% RSLogix 500 project PROC1_COUNTER_RESET_BAK001.RSS, saved by version 8.30.00.16 %
PROJECT "PROC1"    % processor: Bul.1763 MicroLogix 1100 Series B %

PROGRAM FILES
  LAD 2 "MAIN"  2 rungs
  LAD 3 "COUNTERS"  4 rungs

DATA FILES
  O0 OUTPUT  4 elements
  I1 INPUT  6 elements
  S2 STATUS  66 elements
  B3 BINARY  1 elements
  T4 TIMER  1 elements
  C5 COUNTER  1 elements
  R6 CONTROL  1 elements
  N7 INTEGER  1 elements
  F8 FLOAT  1 elements

LADDER 2 "MAIN"
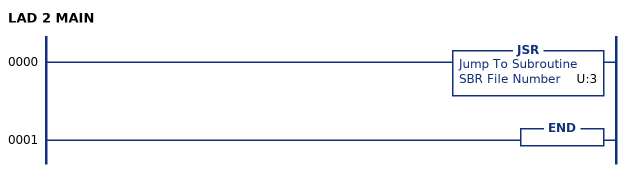
% Rung: 0 %
SOR JSR U:3 EOR
% Rung: 1 %
SOR END EOR

LADDER 3 "COUNTERS"
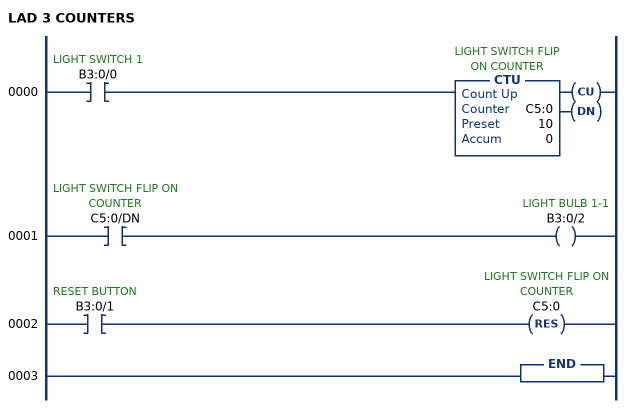
% Rung: 0 %
SOR XIC B3:0/0 CTU C5:0 10 0 EOR
%   B3:0/0  "LIGHT SWITCH 1" %
%   C5:0  "LIGHT SWITCH FLIP ON COUNTER" %
% Rung: 1 %
SOR XIC C5:0/DN OTE B3:0/2 EOR
%   C5:0  "LIGHT SWITCH FLIP ON COUNTER" %
%   B3:0/2  "LIGHT BULB 1-1" %
% Rung: 2 %
SOR XIC B3:0/1 RES C5:0 EOR
%   B3:0/1  "RESET BUTTON" %
%   C5:0  "LIGHT SWITCH FLIP ON COUNTER" %
% Rung: 3 %
SOR END EOR

REVISION NOTES
  0: Added RESET

DATA TABLE (non-zero values as saved)
DATA C5
% .PRE .ACC %
% C5:0 % 10 0
